PROGRAM IntegratorTest
VAR
END_VAR

// NETWORK 1

END_PROGRAM

(* stored: Version 1.1.0.1, ProductVersion 3.1.4024.9
   POU IntegratorTest: Id {472e616a-b374-4df6-a86d-fd7739907b4f}, SpecialFunc None *)
